FUNCTION_BLOCK FB_SingleCoilCylinder EXTENDS FB_UniversalCylinder
VAR_INPUT
	
END_VAR
VAR_OUTPUT
END_VAR
VAR
	(* Coils *)
	poActiveValve	: FB_DigitalOutput;	(* Active position valve function block *)
END_VAR

IF bFirstCycle THEN
	poActiveValve.MR_FirstCycle( sName := CONCAT(sName,':Active_Valve'),sModuleType := ref_poActiveValve.ModuleType, sPortID:= ref_poActiveValve.PortID);
END_IF

SUPER^();

bPositionHold := poActiveValve.Out;

poActiveValve();

METHOD PROTECTED M_SimulationLogic
VAR_INPUT
END_VAR
IF poActiveValve.Out THEN
	piActiveSensor.MR_SetForceValue();
	piHomeSensor.MR_ResetForceValue();
	
ELSIF NOT poActiveValve.Out THEN
	piActiveSensor.MR_ResetForceValue();
	piHomeSensor.MR_SetForceValue();
	
END_IF
END_METHOD

METHOD PROTECTED MS_GoActive
VAR_INPUT
END_VAR
poActiveValve.Out := TRUE;

CASE eCylinderGoActiveState OF
	CYLINDER_MOVE_START_TRACKING:
		piActiveSensor.MR_StartTracking();
		
		IF piActiveSensor.In THEN
			IF TIME_TO_INT(tDelay) = 0 THEN
				eCylinderGoActiveState := CYLINDER_MOVE_DONE;
			ELSE
				eCylinderGoActiveState := CYLINDER_MOVE_DELAY;
			END_IF
		END_IF
		
	CYLINDER_MOVE_DELAY:
		tonGoActiveDelay( IN := TRUE, PT := tDelay);
		
		IF tonGoActiveDelay.Q THEN
			tonGoActiveDelay( IN := FALSE );
			eCylinderGoActiveState := CYLINDER_MOVE_DONE;
		END_IF
		
	CYLINDER_MOVE_DONE:
		eCylinderState := CYLINDER_GO_ACTIVE_DONE;
		
END_CASE
END_METHOD

METHOD PROTECTED MS_GoHome
VAR_INPUT
END_VAR
poActiveValve.Out := FALSE;

CASE eCylinderGoHomeState OF
	CYLINDER_MOVE_START_TRACKING:
		piHomeSensor.MR_StartTracking();
		
		IF piHomeSensor.In THEN
			IF TIME_TO_INT(tDelay) = 0 THEN
				eCylinderGoHomeState := CYLINDER_MOVE_DONE;
			ELSE
				eCylinderGoHomeState := CYLINDER_MOVE_DELAY;
			END_IF
		END_IF
		
	CYLINDER_MOVE_DELAY:
		tonGoHomeDelay( IN := TRUE, PT := tDelay);
		
		IF tonGoHomeDelay.Q THEN
			tonGoHomeDelay( IN := FALSE);
			eCylinderGoHomeState := CYLINDER_MOVE_DONE;
		END_IF
		
	CYLINDER_MOVE_DONE:
		eCylinderState := CYLINDER_GO_HOME_DONE;
	
END_CASE
END_METHOD

METHOD PROTECTED MS_Release
VAR_INPUT
END_VAR
poActiveValve.Out := FALSE;
eCylinderState := CYLINDER_RELEASE_DONE;
END_METHOD

METHOD PROTECTED MS_Reset
VAR_INPUT
END_VAR
poActiveValve.Out := FALSE;

SUPER^.MS_Reset();
END_METHOD

METHOD PROTECTED MS_Uninitialized
poActiveValve.Out := FALSE;
SUPER^.MS_Uninitialized();
END_METHOD

PROPERTY ref_poActiveValve : REFERENCE TO FB_DigitalOutput
GET
ref_poActiveValve REF= poActiveValve;
END_GET
END_PROPERTY

END_FUNCTION_BLOCK

(* stored: Version 1.1.0.1, ProductVersion 3.1.4024.12
   POU FB_SingleCoilCylinder: Id {ff735667-ee11-4b4d-a495-7b30ae1770ad}, SpecialFunc None
   Folder Internal: Id {bd4e0893-441b-42a2-a95f-5fef91e2da12}
   Folder Properties: Id {2f97eea3-808a-4077-8f93-41ec08382c77}
   Folder References: Id {23d4886e-4606-4980-977e-f1da644902f6}
   Folder State Machine: Id {c73d6e29-4e72-4a42-b614-4b720606396c}
   Method M_SimulationLogic: Id {6ed934ea-cdde-413f-86de-c34018e12e8d}
   Method MS_GoActive: Id {8d0c490d-bf7b-4205-bfc2-03ce3373e71e}
   Method MS_GoHome: Id {ad1ecb89-2410-4403-abae-339b747f0278}
   Method MS_Release: Id {f56a5412-390e-4ae3-9608-d8587c79230f}
   Method MS_Reset: Id {c898be4a-5b8b-4afd-bb2e-6c4f162dee35}
   Method MS_Uninitialized: Id {45c5df9f-c2c9-4afb-92fe-f5475ea82beb}
   Property ref_poActiveValve: Id {47f91d18-43e3-40c4-a461-85f571c6b2a9}
   Get Get: Id {ad625b90-ab9e-41f0-b387-99bddf03f929} *)
